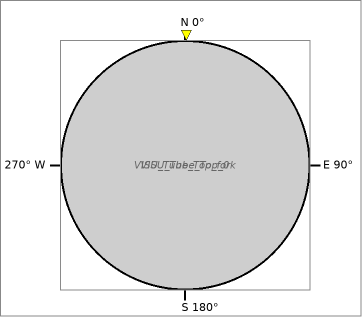
VISUALIZATION VISU_Tube_Top  // 362x317
VAR_IN_OUT
	widget : AxesImageWidget;
END_VAR
    Polyline (185,300) (185,30)
    Polyline (185,295) (185,35)
        p2858320360: widget.mark10Degrees
    Polyline (185,295) (185,35)
        p2858320360: widget.mark10Degrees * 2
    Polyline (185,295) (185,35)
        p2858320360: widget.mark10Degrees * 3
    Polyline (185,295) (185,35)
        p2858320360: widget.mark10Degrees * 4
    Polyline (185,295) (185,35)
        p2858320360: widget.mark10Degrees * 5
    Polyline (185,295) (185,35)
        p2858320360: widget.mark10Degrees * 6
    Polyline (185,295) (185,35)
        p2858320360: widget.mark10Degrees * 7
    Polyline (185,295) (185,35)
        p2858320360: widget.mark10Degrees * 8
    Polyline (185,295) (185,35)
        p2858320360: widget.mark10Degrees * 10
    Polyline (185,295) (185,35)
        p2858320360: widget.mark10Degrees * 11
    Polyline (185,295) (185,35)
        p2858320360: widget.mark10Degrees * 12
    Polyline (185,295) (185,35)
        p2858320360: widget.mark10Degrees * 13
    Polyline (185,295) (185,35)
        p2858320360: widget.mark10Degrees * 14
    Polyline (185,295) (185,35)
        p2858320360: widget.mark10Degrees * 15
    Polyline (185,295) (185,35)
        p2858320360: widget.mark10Degrees * 16
    Polyline (185,295) (185,35)
        p2858320360: widget.mark10Degrees * 17
    Polyline (50,165) (320,165)
    Ellipse (60,40 250x250)
    Frame (60,40 250x250)
        shows VISU_Tube_Top_fork(azi := widget.azi)
    Frame (60,40 250x250), frame switch variable: widget.aziTopTubShown
        shows VISU_Tube_Top_0(azi := widget.azi)
        shows VISU_Tube_Top_1(azi := widget.azi)
        shows VISU_Tube_Top_2(azi := widget.azi)
        shows VISU_Tube_Top_3(azi := widget.azi)
        shows VISU_Tube_Top_4(azi := widget.azi)
        shows VISU_Tube_Top_5(azi := widget.azi)
        shows VISU_Tube_Top_6(azi := widget.azi)
        shows VISU_Tube_Top_7(azi := widget.azi)
        shows VISU_Tube_Top_8(azi := widget.azi)
        shows VISU_Tube_Top_9(azi := widget.azi)
        shows VISU_Tube_Top_10(azi := widget.azi)
        shows VISU_Tube_Top_11(azi := widget.azi)
        shows VISU_Tube_Top_12(azi := widget.azi)
        shows VISU_Tube_Top_13(azi := widget.azi)
        shows VISU_Tube_Top_14(azi := widget.azi)
    Rectangle (320,155 40x20), "E 90°"
    Rectangle (0,155 50x20), "270° W"
    Rectangle (175,15 35x15), "N 0°"
    Rectangle (175,300 50x15), "S 180°"
    Polygon (181,30) (186,40) (191,30), invisible if: widget.aziTargetInvisible
        p2858320360: widget.aziTarget
END_VISUALIZATION

(* stored: Version 1.1.0.1, ProductVersion 3.1.4019.2
   Visu VISU_Tube_Top: Id {f83e5e6b-b9bb-4a45-aaaa-a155c1295d6e} *)
